(* Logix 5000 project; controller Y059_LHM vendor 1 type 14 code 156 rev 32.13; software revision 32.00; part 2 of 2 *)

VAR_GLOBAL   (* controller tags *)
   FromDeltaV_HeartBeat : DINT := 58;   // From DeltaV Heartbeat DINT
   FromDeltaV_PumpAFaultReset : BOOL;   // From DeltaV Pump A Fault Reset
   FromDeltaV_PumpARun : BOOL;   // From DeltaV Pump A Run Command
   FromDeltaV_PumpASpd : REAL := 5.0;   // From DeltaV Pump A Speed
   FromDeltaV_PumpBFaultReset : BOOL;   // From DeltaV Pump B Fault Reset
   FromDeltaV_PumpBRun : BOOL;   // From DeltaV Pump B Run Command
   FromDeltaV_PumpBSpd : REAL := 5.0;   // From DeltaV Pump B Speed
   FromDeltaV_PumpCFaultReset : BOOL;   // From DeltaV Pump C Fault Reset
   FromDeltaV_PumpCRun : BOOL;   // From DeltaV Pump C Run Command
   FromDeltaV_PumpCSpd : REAL;   // From DeltaV Pump C Speed
   Motion_Pumps : MOTION_GROUP;   // Run Command & Speed From DeltaV
   PumpA_LocalFault : BOOL;
   PumpB_LocalFault : BOOL;
   PumpC_LocalFault : BOOL;
   SIC_101_Axis : AXIS_CIP_DRIVE;
   SIC_201_Axis : AXIS_CIP_DRIVE;
   ToDeltaV_Bool : BOOL[32] := ([1] := 1, [9] := 1, [26] := 1);
        [25]   // isColumnPressureHigh
        [26]   // isEstopResetNeeded
        [16]   // Pump C isDecontacted
        [8]   // Pump B isDecontacted
        [2]   // Pump A isPressureHigh
        [3]   // Pump A isRunning
        [17]   // Pump C isFault
        [18]   // Pump C isPressureHigh
        [4]   // Pump A isServoOk
        [19]   // Pump C isRunning
        [20]   // Pump C isServoOK
        [23]   // isDeltaV_HeartBeat_Error
        [1]   // Pump A isFault
        [9]   // Pump B isFault
        [10]   // Pump B isPressureHigh
        [24]   // isEstopEngaged
        [11]   // Pump B isRunning
        [12]   // Pump B isServoOK
        [0]   // Pump A isDecontacted
   ToDeltaV_DINT : DINT[8] := ([3] := 61);
        [3]   // Heart Beat
        [0]   // Pump A Fault Code
        [1]   // Pump B Fault Code
        [2]   // Pump C Fault Code
        [4]   // Pump A Fault Type
        [5]   // Pump B Fault Type
        [6]   // Pump C Fault Type
   ToDeltaV_Real : REAL[8] := ([3] := 50.0);
        [0]   // Pump A Speed Feedback
        [1]   // Pump A Speed Setpoint
        [2]   // Pump B Speed Feedback
        [3]   // Pump B Speed Setpoint
        [4]   // Pump C Speed Feedback
        [5]   // Pump C Speed Setpoint
END_VAR

PROGRAM MainProgram   (* main routine Routine_Main, fault routine FaultRoutine *)
VAR
   ArrayOverrun : BOOL;
   DeltaV_HB_Prev : DINT := 58;
   DeltaV_HB_TimeoutTime : REAL := 5.0;   // DeltaV Heart Beat Time out Time (default 30 second)
   DeltaV_HB_Timer : TIMER := (PRE := 5000, ACC := 4600, EN := 1, TT := 1);   // DeltaV Heart Beat Monitor Timer
   FaultCode_Sic_101 : ServoFaultCode := (DriveConnStatus := 16#0000_3000);
   FaultCode_Sic_201 : ServoFaultCode := (DriveConnStatus := 16#0000_3000);
   HeartBeatErrorLatch : BOOL;   // Latch when deltaV Heart Beat error
   HeartBeatTimer : TIMER := (PRE := 1000, ACC := 1000, EN := 1, DN := 1);   // PLC Heart Beat Timer
   Local_PumpA : PumpController := (isFaulted := 1, SpeedSP.Max := 100.0, SpeedFeedback.Max := 100.0, Ok2Run := 1, ResetTimer.PRE := 10000);
   Local_PumpB : PumpController := (isFaulted := 1, SpeedSP.SP := 50.0, SpeedSP.Max := 100.0, SpeedFeedback.Max := 100.0, Ok2Run := 1, ResetTimer.PRE := 10000);
   Local_PumpC : PumpController := (Ok2Run := 1);
   Major_Fault_Record : FaultRecord;
   Proc_Sic_101 : SERVO_AOI := (GearBox_Ratio := 6.25, Axis_AccDec := 20.0, Pump_RPM_Max := 287);
   Proc_Sic_201 : SERVO_AOI := (GearBox_Ratio := 6.25, Axis_AccDec := 20.0, Pump_RPM_Max := 287);
   Proc_Sic_301 : SERVO_AOI := (GearBox_Ratio := 10.0, Axis_AccDec := 20.0, Pump_RPM_Max := 173, Pump_RPM_Val := 30.88, Motor_RPS := 5.1466665);
   ProcedureEnable : DINT := 255;
   PumpA_DriveConnStat : DINT := 12288;
   PumpB_DriveConnStat : DINT := 12288;
   TrapFaults : BOOL := 1;
END_VAR

ROUTINE Exchange_FromPumpTags   (* ladder *)
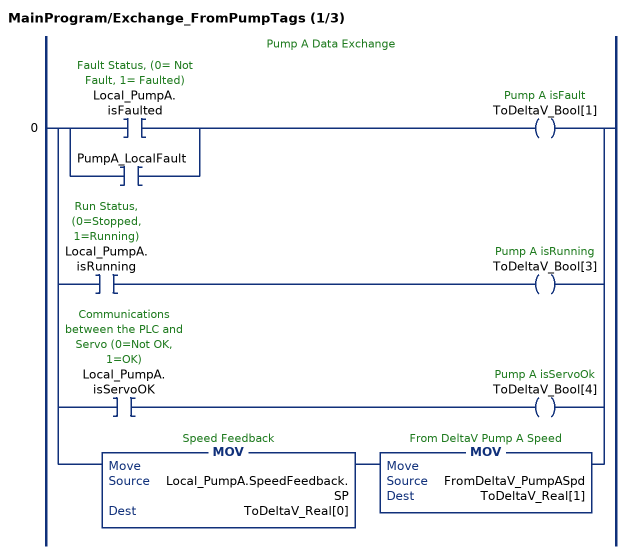
   // Pump A Data Exchange
   0: [[XIC(Local_PumpA.isFaulted) ,XIC(PumpA_LocalFault) ] OTE(ToDeltaV_Bool[1]) ,XIC(Local_PumpA.isRunning) OTE(ToDeltaV_Bool[3]) ,XIC(Local_PumpA.isServoOK) OTE(ToDeltaV_Bool[4]) ,MOV(Local_PumpA.SpeedFeedback.SP,ToDeltaV_Real[0]) MOV(FromDeltaV_PumpASpd,ToDeltaV_Real[1]) ];
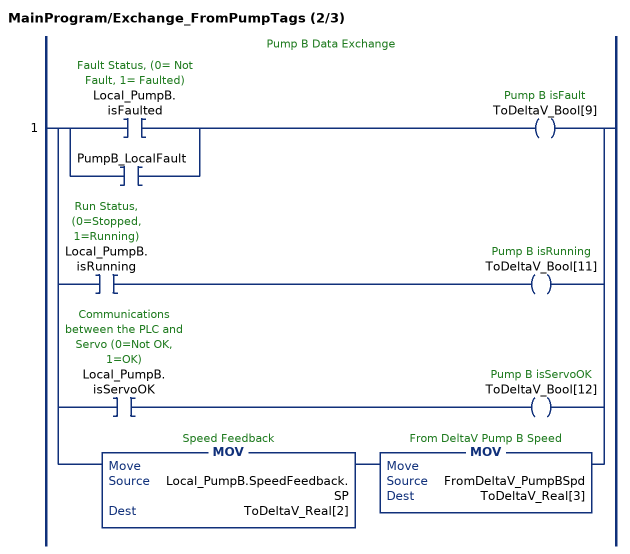
   // Pump B Data Exchange
   1: [[XIC(Local_PumpB.isFaulted) ,XIC(PumpB_LocalFault) ] OTE(ToDeltaV_Bool[9]) ,XIC(Local_PumpB.isRunning) OTE(ToDeltaV_Bool[11]) ,XIC(Local_PumpB.isServoOK) OTE(ToDeltaV_Bool[12]) ,MOV(Local_PumpB.SpeedFeedback.SP,ToDeltaV_Real[2]) MOV(FromDeltaV_PumpBSpd,ToDeltaV_Real[3]) ];
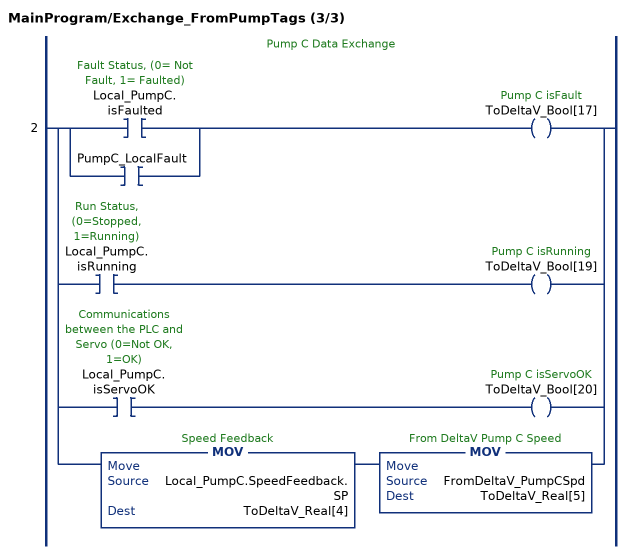
   // Pump C Data Exchange
   2: [[XIC(Local_PumpC.isFaulted) ,XIC(PumpC_LocalFault) ] OTE(ToDeltaV_Bool[17]) ,XIC(Local_PumpC.isRunning) OTE(ToDeltaV_Bool[19]) ,XIC(Local_PumpC.isServoOK) OTE(ToDeltaV_Bool[20]) ,MOV(Local_PumpC.SpeedFeedback.SP,ToDeltaV_Real[4]) MOV(FromDeltaV_PumpCSpd,ToDeltaV_Real[5]) ];
END_ROUTINE

ROUTINE Exchange_ToPumpTags   (* ladder *)
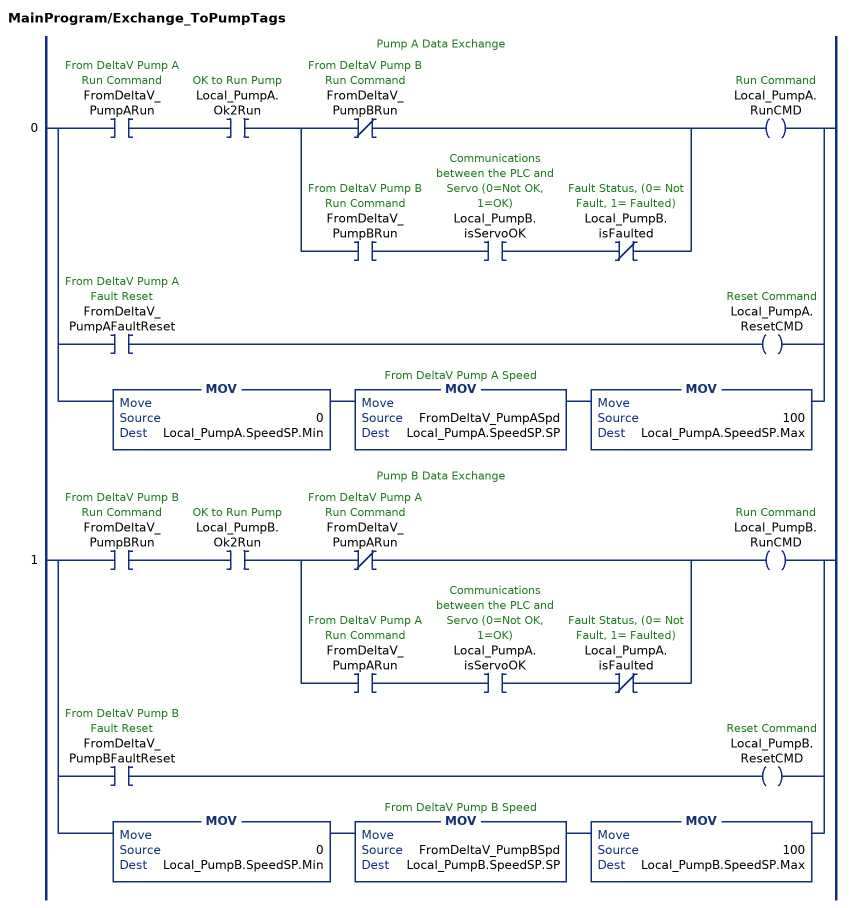
   // Pump A Data Exchange
   0: [XIC(FromDeltaV_PumpARun) XIC(Local_PumpA.Ok2Run) [XIO(FromDeltaV_PumpBRun) ,XIC(FromDeltaV_PumpBRun) XIC(Local_PumpB.isServoOK) XIO(Local_PumpB.isFaulted) ] OTE(Local_PumpA.RunCMD) ,XIC(FromDeltaV_PumpAFaultReset) OTE(Local_PumpA.ResetCMD) ,MOV(0,Local_PumpA.SpeedSP.Min) MOV(FromDeltaV_PumpASpd,Local_PumpA.SpeedSP.SP) MOV(100,Local_PumpA.SpeedSP.Max) ];
   // Pump B Data Exchange
   1: [XIC(FromDeltaV_PumpBRun) XIC(Local_PumpB.Ok2Run) [XIO(FromDeltaV_PumpARun) ,XIC(FromDeltaV_PumpARun) XIC(Local_PumpA.isServoOK) XIO(Local_PumpA.isFaulted) ] OTE(Local_PumpB.RunCMD) ,XIC(FromDeltaV_PumpBFaultReset) OTE(Local_PumpB.ResetCMD) ,MOV(0,Local_PumpB.SpeedSP.Min) MOV(FromDeltaV_PumpBSpd,Local_PumpB.SpeedSP.SP) MOV(100,Local_PumpB.SpeedSP.Max) ];
END_ROUTINE

ROUTINE FaultRoutine   (* ladder *)
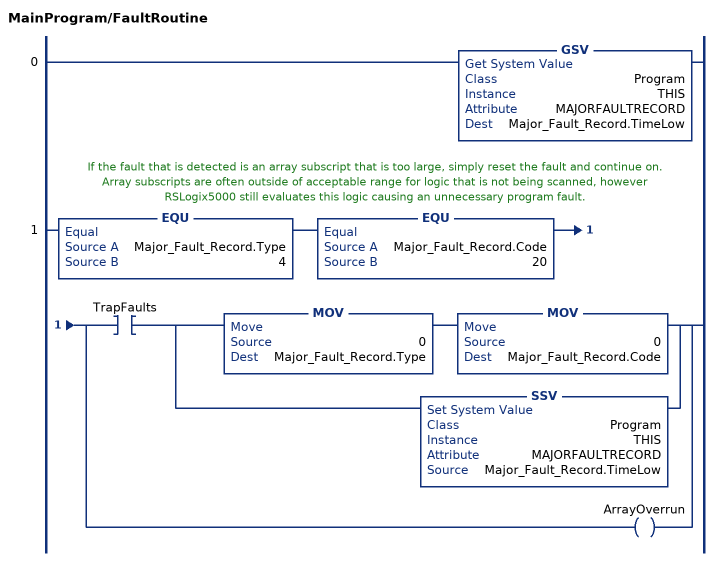
   0: GSV(Program,THIS,MAJORFAULTRECORD,Major_Fault_Record.TimeLow);
   // If the fault that is detected is an array subscript that is too large, simply reset the fault and continue on.
   // Array subscripts are often outside of acceptable range for logic that is not being scanned, however RSLogix5000 still evaluates this logic causing an unnecessary program fault.
   1: EQU(Major_Fault_Record.Type,4)EQU(Major_Fault_Record.Code,20)[XIC(TrapFaults) [MOV(0,Major_Fault_Record.Type) MOV(0,Major_Fault_Record.Code) ,SSV(Program,THIS,MAJORFAULTRECORD,Major_Fault_Record.TimeLow) ] ,OTE(ArrayOverrun) ];
END_ROUTINE

ROUTINE Routine_HeartBeat   (* ladder *)
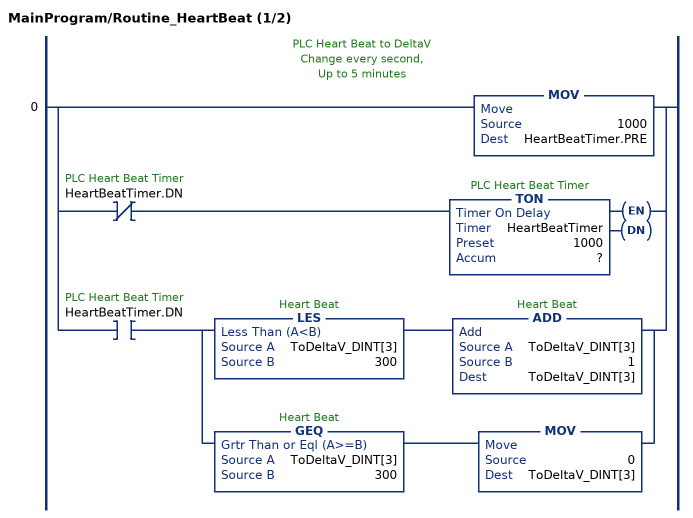
   // PLC Heart Beat to DeltaV
   // Change every second,
   // Up to 5 minutes
   0: [MOV(1000,HeartBeatTimer.PRE) ,XIO(HeartBeatTimer.DN) TON(HeartBeatTimer,?,?) ,XIC(HeartBeatTimer.DN) [LES(ToDeltaV_DINT[3],300) ADD(ToDeltaV_DINT[3],1,ToDeltaV_DINT[3]) ,GEQ(ToDeltaV_DINT[3],300) MOV(0,ToDeltaV_DINT[3]) ] ];
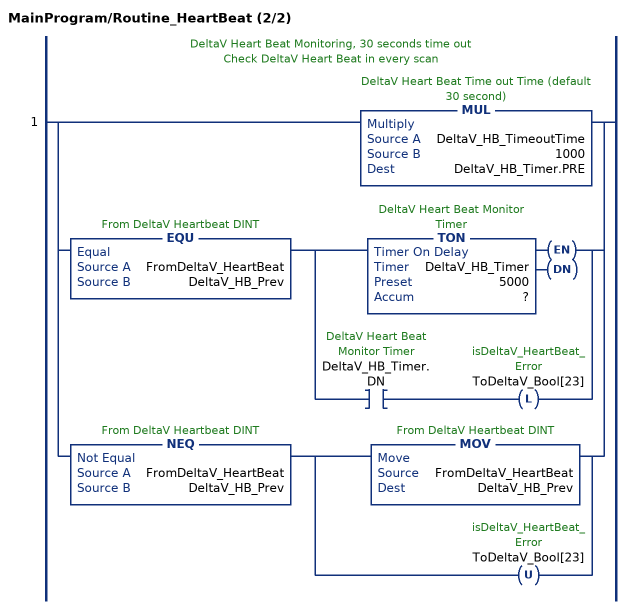
   // DeltaV Heart Beat Monitoring, 30 seconds time out
   // Check DeltaV Heart Beat in every scan
   1: [MUL(DeltaV_HB_TimeoutTime,1000,DeltaV_HB_Timer.PRE) ,EQU(FromDeltaV_HeartBeat,DeltaV_HB_Prev) [TON(DeltaV_HB_Timer,?,?) ,XIC(DeltaV_HB_Timer.DN) OTL(ToDeltaV_Bool[23]) ] ,NEQ(FromDeltaV_HeartBeat,DeltaV_HB_Prev) [MOV(FromDeltaV_HeartBeat,DeltaV_HB_Prev) ,OTU(ToDeltaV_Bool[23]) ] ];
END_ROUTINE

ROUTINE Routine_Main   (* ladder *)
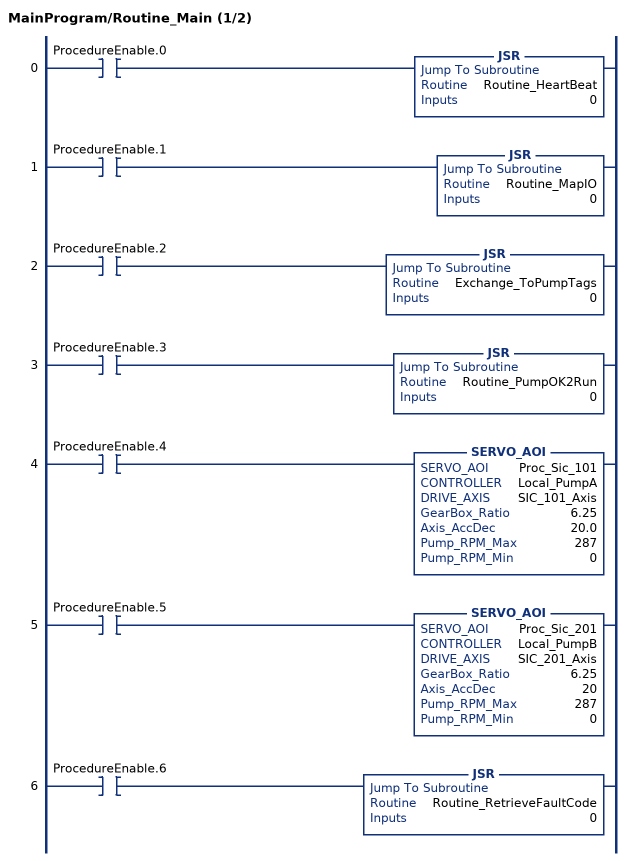
   0: XIC(ProcedureEnable.0)JSR(Routine_HeartBeat,0);
   1: XIC(ProcedureEnable.1)JSR(Routine_MapIO,0);
   2: XIC(ProcedureEnable.2)JSR(Exchange_ToPumpTags,0);
   3: XIC(ProcedureEnable.3)JSR(Routine_PumpOK2Run,0);
   4: XIC(ProcedureEnable.4)SERVO_AOI(Proc_Sic_101,Local_PumpA,SIC_101_Axis,6.25,20.0,287,0);
   5: XIC(ProcedureEnable.5)SERVO_AOI(Proc_Sic_201,Local_PumpB,SIC_201_Axis,6.25,20,287,0);
   6: XIC(ProcedureEnable.6)JSR(Routine_RetrieveFaultCode,0);
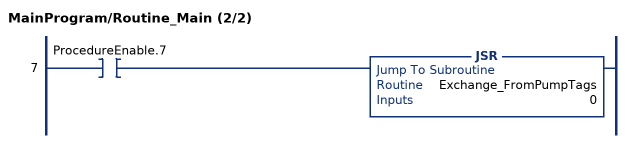
   7: XIC(ProcedureEnable.7)JSR(Exchange_FromPumpTags,0);
END_ROUTINE

ROUTINE Routine_MapIO   (* structured text *)
   // IO Mapping
   
   //*********** Module 1 ***********
   //********** 1769-IQ16 ***********
   
   ToDeltaV_Bool[2] := Local:1:I.Data.0; 							// PSH-7355A (Pump A isPressureHigh)
   ToDeltaV_Bool[10] := Local:1:I.Data.1; 							// PSH-7355B (Pump B isPressureHigh)
   ToDeltaV_Bool[25] := Local:1:I.Data.2; 							// Column Pressure High (isColumnPressureHigh)
   ToDeltaV_Bool[18] := Local:1:I.Data.3; 							// FuturePumpSTOStatus (Pump C isPressureHigh)
   ToDeltaV_Bool[26] := Local:1:I.Data.4;							// Master Reset (isESTOPResetNeeded)
   ToDeltaV_Bool[24] := Local:1:I.Data.5;  						// Emergency Stop Push Button (isEStopEngaged)
   ToDeltaV_Bool[0] := Local:1:I.Data.6;  							// 7355 D-Con/High Temp (Pump A isDecontacted)
   ToDeltaV_Bool[8]:= Local:1:I.Data.7;  							// 7355 B-Con/High Temp (Pump B isDecontacted)
   //Not Used := Local:1:I.Data.8; 								// 7355-AA
   //Not Used := Local:1:I.Data.9; 								// 7355-AB
   //Not Used := Local:1:I.Data.10; 								// 7355-AC
   //Not Used := Local:1:I.Data.11; 								// 7355-BA
   //Not Used := Local:1:I.Data.12; 								// 7355-BB
   //Not Used := Local:1:I.Data.13;								// 7355-BC
   //Spare := Local:1:I.Data.14; 									// Spare
   //Spare := Local:1:I.Data.15; 									// Spare
   
   
   
   //*********** Module 2 ***********
   //*********** 1769-OB16 **********
   
   Local:2:O.Data.0 := FromDeltaV_PumpAFaultReset OR FromDeltaV_PumpBFaultReset OR FromDeltaV_PumpCFaultReset;		//STO Reset
   Local:2:O.Data.1 := FromDeltaV_PumpAFaultReset OR FromDeltaV_PumpBFaultReset OR FromDeltaV_PumpCFaultReset;		// Emergency Stop Reset
   //Local:2:O.Data.2 := Spare;									// Spare
   //Local:2:O.Data.3 := Spare;									// Spare
   //Local:2:O.Data.4 := Spare;									// Spare
   //Local:2:O.Data.5 := Spare;									// Spare
   //Local:2:O.Data.6 := Spare;									// Spare
   //Local:2:O.Data.7 := Spare;									// Spare
   //Local:2:O.Data.8 := Spare;									// Spare
   //Local:2:O.Data.9 := Spare;									// Spare
   //Local:2:O.Data.10 := Spare;									// Spare
   //Local:2:O.Data.11 := Spare;									// Spare
   //Local:2:O.Data.12 := Spare;									// Spare
   //Local:2:O.Data.13 := Spare;									// Spare
   //Local:2:O.Data.14 := Spare;									// Spare
   //Local:2:O.Data.15 := Spare;									// Spare
   
END_ROUTINE

ROUTINE Routine_PumpOK2Run   (* ladder *)
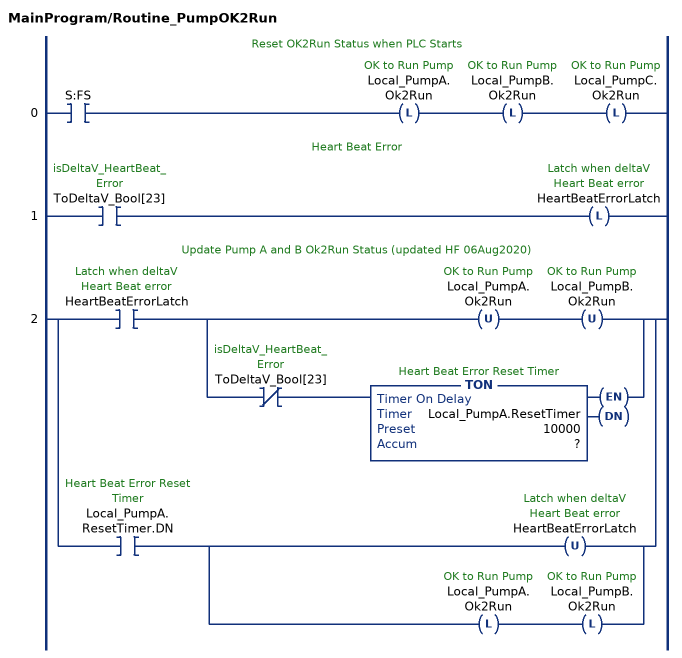
   // Reset OK2Run Status when PLC Starts
   0: XIC(S:FS)OTL(Local_PumpA.Ok2Run)OTL(Local_PumpB.Ok2Run)OTL(Local_PumpC.Ok2Run);
   // Heart Beat Error
   1: XIC(ToDeltaV_Bool[23])OTL(HeartBeatErrorLatch);
   // Update Pump A and B Ok2Run Status (updated HF 06Aug2020)
   2: [XIC(HeartBeatErrorLatch) [OTU(Local_PumpA.Ok2Run) OTU(Local_PumpB.Ok2Run) ,XIO(ToDeltaV_Bool[23]) TON(Local_PumpA.ResetTimer,?,?) ] ,XIC(Local_PumpA.ResetTimer.DN) [OTU(HeartBeatErrorLatch) ,OTL(Local_PumpA.Ok2Run) OTL(Local_PumpB.Ok2Run) ] ];
END_ROUTINE

ROUTINE Routine_RetrieveFaultCode   (* ladder *)
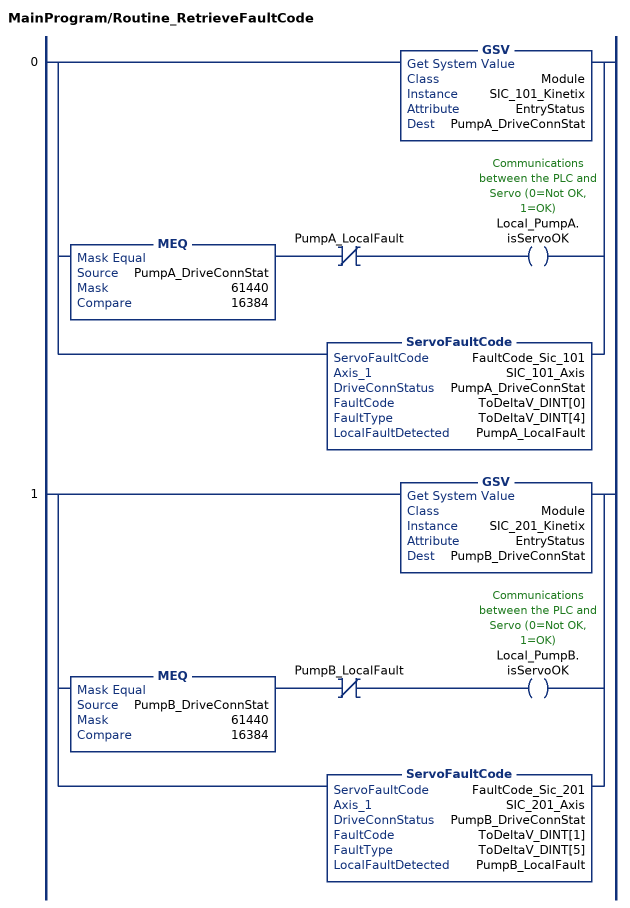
   0: [GSV(Module,SIC_101_Kinetix,EntryStatus,PumpA_DriveConnStat) ,MEQ(PumpA_DriveConnStat,61440,16384) XIO(PumpA_LocalFault) OTE(Local_PumpA.isServoOK) ,ServoFaultCode(FaultCode_Sic_101,SIC_101_Axis,PumpA_DriveConnStat,ToDeltaV_DINT[0],ToDeltaV_DINT[4],PumpA_LocalFault) ];
   1: [GSV(Module,SIC_201_Kinetix,EntryStatus,PumpB_DriveConnStat) ,MEQ(PumpB_DriveConnStat,61440,16384) XIO(PumpB_LocalFault) OTE(Local_PumpB.isServoOK) ,ServoFaultCode(FaultCode_Sic_201,SIC_201_Axis,PumpB_DriveConnStat,ToDeltaV_DINT[1],ToDeltaV_DINT[5],PumpB_LocalFault) ];
END_ROUTINE
END_PROGRAM
